FUNCTION_BLOCK FB_LABEL (* GUI label *)
  (* Standard: 61499-1; ApplicationDomain: GUI; Function: Label *)
  (* Version 0.1, 2002-05-03, JHC, Rockwell Automation, Made QI initial value = true. *)
  (* Version 0.0, 2001-03-04, JHC, Rockwell Automation, Updated documentation. *)
  (* Compiler header: package fb.rt.hmi; import fb.rt.*; import java.awt.*; *)
  (* Compiler Java IBM VisualAge 3.0 *)
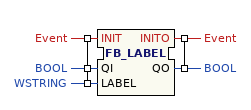
  EVENT_INPUT
    INIT WITH QI, LABEL; (* Service Initialization *)
  END_EVENT
  EVENT_OUTPUT
    INITO WITH QO; (* Initialization Confirm *)
  END_EVENT
  VAR_INPUT
    QI : BOOL := true;
    LABEL : WSTRING; (* Label *)
  END_VAR
  VAR_OUTPUT
    QO : BOOL;
  END_VAR
  SERVICE FB_LABEL/Label
    SEQUENCE normal_establishment
      FB_LABEL.INIT+(LABEL) -> Label.setText(LABEL) -> FB_LABEL.INITO+();
    END_SEQUENCE
    SEQUENCE normal_termination
      FB_LABEL.INIT-() -> FB_LABEL.INITO-();
    END_SEQUENCE
  END_SERVICE
END_FUNCTION_BLOCK
